(* PLC project Unnamed, Unknown Unnamed 1 *)
(* stored: creationDateTime 2025-10-15T14:42:18, modificationDateTime 2025-10-31T16:00:33 *)

(* Infeed & Conveying *)
PROGRAM program1
  VAR
    EStop AT %IX1.0 : BOOL;
    Bottle_Jam AT %IX1.1 : BOOL;  (* Sensor that monitors bottle jam. *)
    Speed_Encoder AT %IX1.2 : BOOL;  (* Conveyor speed encoder. *)
    Speed_Control AT %IX1.3 : BOOL;  (* Speed control input. *)
    Conveyor_Enable AT %MX1.0 : BOOL;  (* Memory for enabling conveyor output. *)
    Conveyor_Motor AT %QX1.0 : BOOL;  (* Conveyor motor output. *)
    Alarm_Jam AT %QX1.1 : BOOL;  (* Alarm that sounds when jam occurs. *)
    Conveyor_Speed_Command AT %QX1.2 : BOOL;  (* Output command that controls conveyor speed. *)
    Line_Light_Tower AT %QX1.3 : BOOL;  (* Indicator light for conveyor status. *)
  END_VAR

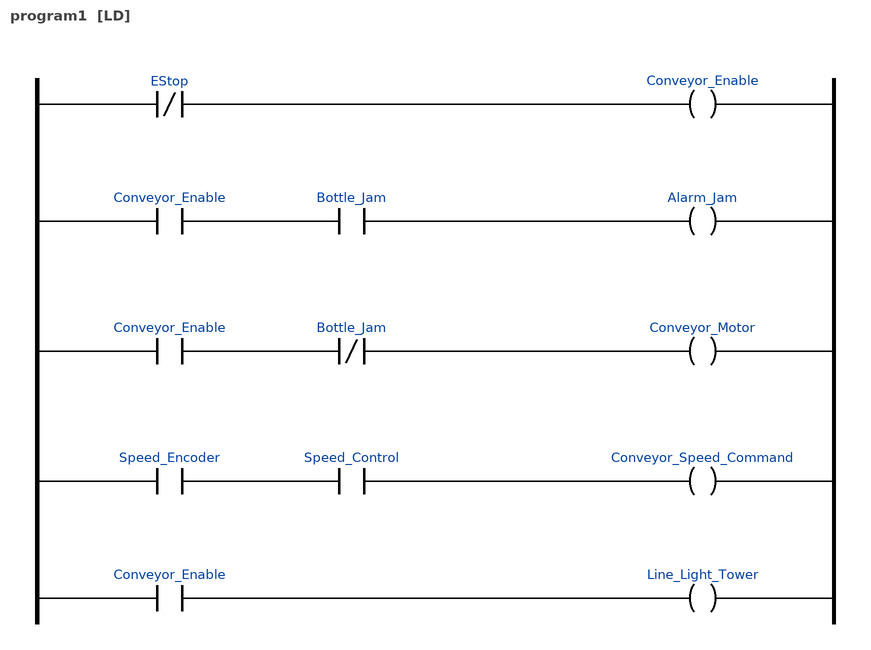
(* LD diagram, written out as Structured Text *)
Conveyor_Enable := NOT EStop;
Alarm_Jam := Conveyor_Enable AND Bottle_Jam;
Conveyor_Motor := Conveyor_Enable AND NOT Bottle_Jam;
Conveyor_Speed_Command := Speed_Encoder AND Speed_Control;
Line_Light_Tower := Conveyor_Enable;
END_PROGRAM

(* Bottle Positioning & Detection *)
PROGRAM program2
  VAR
    Switch_Conveyor AT %IX2.0 : BOOL;  (* Input switch that designates conveyor can start. *)
    Bottle_Presence_Fill AT %IX2.1 : BOOL;  (* Input that designates bottle is at filling station. *)
    Bottle_Presence_Cap AT %IX2.2 : BOOL;  (* Input that designates bottle is at capping station. *)
    Bottle_Presence_Label AT %IX2.3 : BOOL;  (* Input that designates bottle is at labeling station. *)
    Stop_Conveyor_Fill AT %MX2.0 : BOOL;  (* Stop the conveyor at the filling station. *)
    Stop_Conveyor_Cap AT %MX2.1 : BOOL;  (* Stop the conveyor at the capping station. *)
    Stop_Conveyor_Label AT %MX2.2 : BOOL;  (* Stop the conveyor at the labeling station. *)
    Conveyor_Enable AT %QX2.0 : BOOL;  (* Conveyor output. *)
  END_VAR

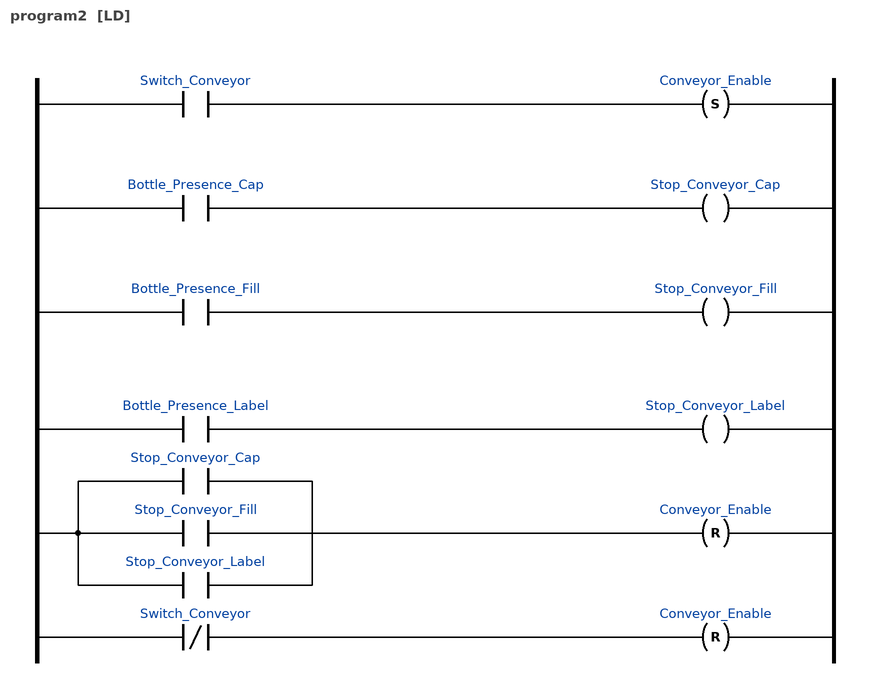
(* LD diagram, written out as Structured Text *)
Stop_Conveyor_Cap := Bottle_Presence_Cap;
Stop_Conveyor_Fill := Bottle_Presence_Fill;
Stop_Conveyor_Label := Bottle_Presence_Label;
IF Stop_Conveyor_Cap OR Stop_Conveyor_Fill OR Stop_Conveyor_Label THEN Conveyor_Enable := FALSE; END_IF;
IF Switch_Conveyor THEN Conveyor_Enable := TRUE; END_IF;
IF NOT Switch_Conveyor THEN Conveyor_Enable := FALSE; END_IF;
END_PROGRAM

(* Filling Subsystem *)
PROGRAM program3
  VAR
    Bottle_Presence_Fill AT %IX3.0 : BOOL;  (* Input that designates bottle is at filling station. *)
    Optical_Neck_Sensor AT %IX3.1 : BOOL;  (* Input that checks if bottle is okay to fill. *)
    Fill_Timer AT %IX3.2 : BOOL;  (* Input timer that tells system how long to fill bottle to full. *)
    Fill_Flowrate AT %IX3.3 : BOOL;  (* Input sensor that monitors flowrate into bottle. *)
    Fill_Temperature AT %IX3.4 : BOOL;  (* Input sensor that monitors temperature of liquid into bottle. *)
    Fill_Enable AT %MX3.0 : BOOL;  (* Memory that stores if its okay to fill. *)
    Fill_Valve AT %QX3.0 : BOOL;  (* Output fill valve. *)
    Fill_Pump_Speed AT %QX3.1 : BOOL;  (* Output fill pump speed. *)
    Fill_Alarm AT %QX3.2 : BOOL;  (* Alarm that sounds when bottle fill goes wrong. *)
  END_VAR

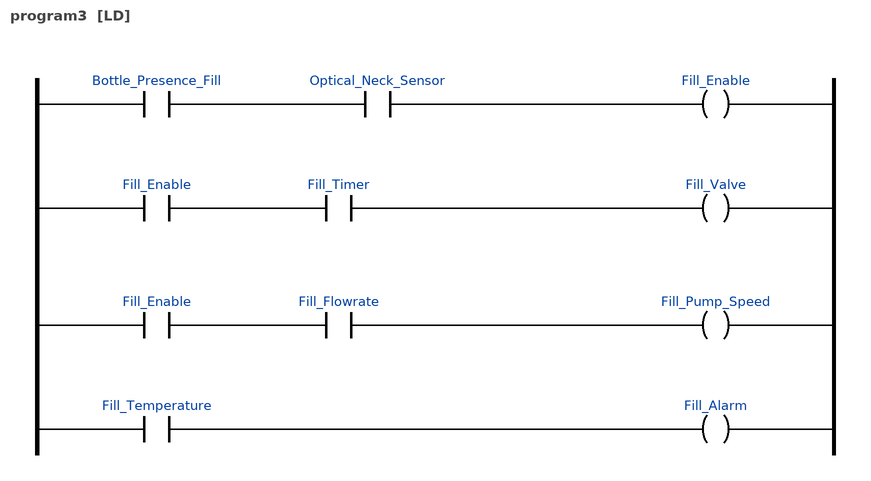
(* LD diagram, written out as Structured Text *)
Fill_Enable := Bottle_Presence_Fill AND Optical_Neck_Sensor;
Fill_Valve := Fill_Enable AND Fill_Timer;
Fill_Pump_Speed := Fill_Enable AND Fill_Flowrate;
Fill_Alarm := Fill_Temperature;
END_PROGRAM

(* Pump & Fluid Utilities *)
PROGRAM program4
  VAR
    Min_Tank_Level AT %IX4.0 : BOOL;  (* Input that arbitrates the minimum tank level. *)
    Prssure_Pump AT %IX4.1 : BOOL;  (* Input that acts as a pressure control. *)
    Pump_Enable AT %MX4.0 : BOOL;  (* Memory that stores if its okay to pump. *)
    Fill_Pump_Speed AT %QX4.0 : BOOL;  (* Output fill pump speed. *)
    Tank_Alarm AT %QX4.1 : BOOL;  (* Alarm that sounds when tank is not at optimal conditions. *)
  END_VAR

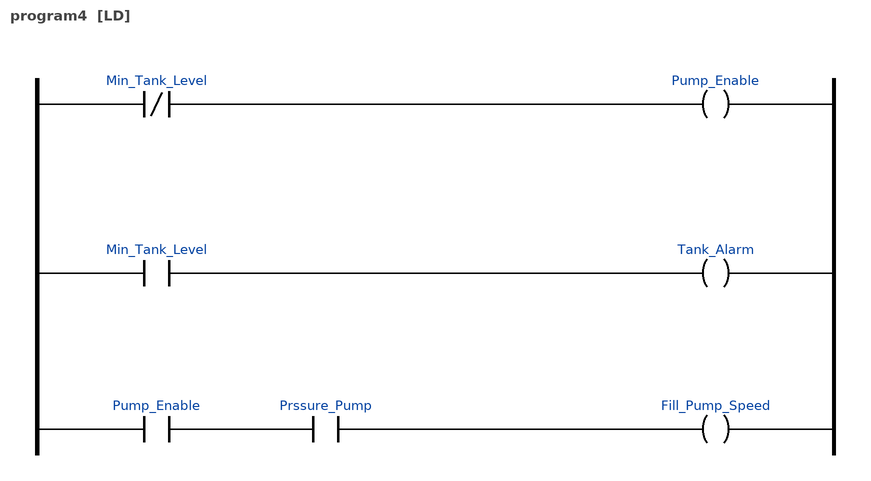
(* LD diagram, written out as Structured Text *)
Pump_Enable := NOT Min_Tank_Level;
Fill_Pump_Speed := Pump_Enable AND Prssure_Pump;
Tank_Alarm := Min_Tank_Level;
END_PROGRAM

PROGRAM program5
  VAR
    Min_Cap_Hopper_Level AT %IX5.0 : BOOL;  (* Input that determines if the cap level within the hopper is above the minium allowed amount *)
    Cap_Presence_Hopper AT %IX5.1 : BOOL;  (* Input that designates a cap is at the hopper *)
    Min_Cap_Torque_Sensor AT %IX5.2 : BOOL;  (* Input that determines if the cap torque sensor is within maximum specification *)
    Max_Cap_Torque_Sensor AT %IX5.3 : BOOL;  (* Input that determines if the cap torque sensor is within minimum specification *)
    Capping_Enable AT %MX5.0 : BOOL;  (* Memory that stores if it is okay to cap *)
    Alarm_Caps AT %QX5.1 : BOOL;  (* Alarm to notify that cap hopper level is low *)
    Cap_Bottle AT %QX5.2 : BOOL;  (* Output Capping Bottle *)
    Actuator_Alarm AT %QX5.3 : BOOL;  (* Alarm to notify if the actuator is out of specification *)
  END_VAR

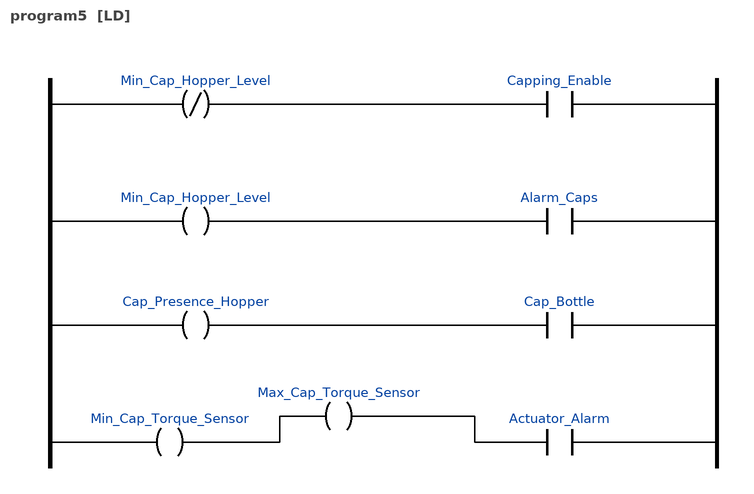
(* LD diagram, written out as Structured Text *)
Cap_Presence_Hopper := TRUE;
Min_Cap_Hopper_Level := NOT TRUE;
Min_Cap_Hopper_Level := TRUE;
Min_Cap_Torque_Sensor := TRUE;
Max_Cap_Torque_Sensor := TRUE;
(* drawn but not wired to any output: Capping_Enable, Alarm_Caps, Cap_Bottle, Actuator_Alarm *)
END_PROGRAM

PROGRAM program6
  VAR
    Bottle_Presence_Label AT %IX6.0 : BOOL;  (* Input that designates a bottle is at the labeling station *)
    Label_Presence AT %IX6.1 : BOOL;  (* Input that indicates a label is present at the labeling station *)
    Label_Positioning AT %IX6.2 : BOOL;  (* Input that checks the positioning of the label to ensure it is applied properly *)
    Label_Applicator AT %QX6.0 : BOOL;  (* Output for application of the label on to the bottle *)
    Actuator_Alarm AT %QX6.1 : BOOL;  (* Alarm to notify if the actuator is out of specification *)
  END_VAR

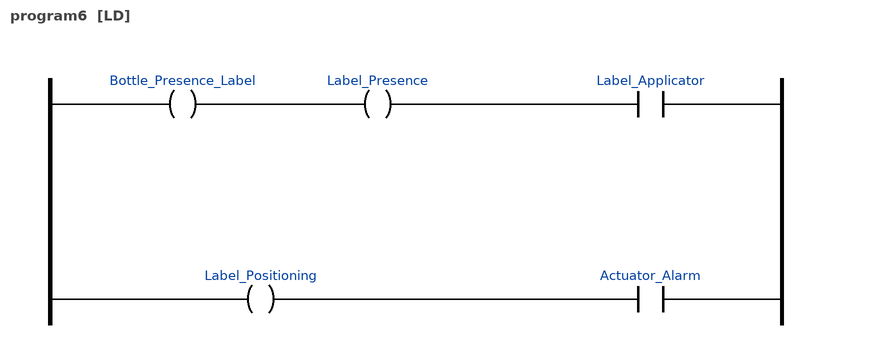
(* LD diagram, written out as Structured Text *)
Bottle_Presence_Label := TRUE;
Label_Presence := TRUE;
Label_Positioning := TRUE;
(* drawn but not wired to any output: Label_Applicator, Actuator_Alarm *)
END_PROGRAM

PROGRAM program7
  VAR
    Fill_Level_Detect AT %IX7.0 : BOOL;  (* Input to detect the level that the bottle has been filled to to ensure it is within specification *)
    Optical_Neck_sensor AT %IX7.1 : BOOL;  (* Input to detect the condition of the neck, ensuring there are no cracks or damage present on the bottle neck *)
    Bottle_Weight AT %IX7.2 : BOOL;  (* Input to detect the weight of the bottle does not exceed the threshold *)
    Cap_Torque_Sensor AT %IX7.3 : BOOL;  (* Input to detect the cap is not overtorqued *)
    Reject_Bottle AT %QX7.0 : BOOL;  (* Output to reject bottle if any of the inputs detect faults *)
  END_VAR

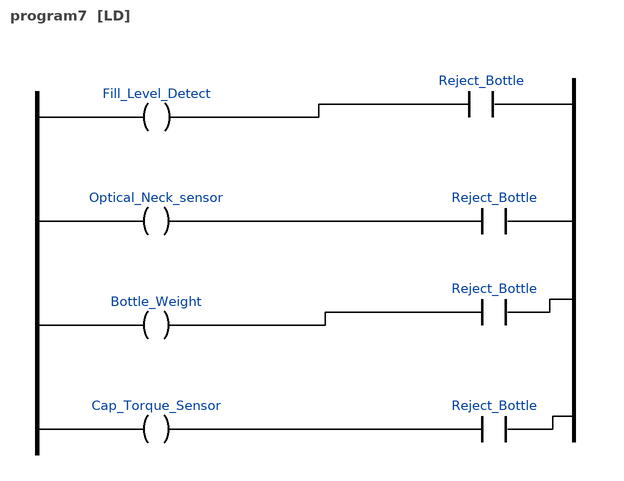
(* LD diagram, written out as Structured Text *)
Fill_Level_Detect := TRUE;
Optical_Neck_sensor := TRUE;
Bottle_Weight := TRUE;
Cap_Torque_Sensor := TRUE;
(* drawn but not wired to any output: Reject_Bottle, Reject_Bottle, Reject_Bottle, Reject_Bottle *)
END_PROGRAM

CONFIGURATION Config0
  RESOURCE Res0 ON PLC
    TASK task1(INTERVAL := T#20ms, PRIORITY := 0);
    TASK task2(INTERVAL := T#20ms, PRIORITY := 0);
    TASK task3(INTERVAL := T#20ms, PRIORITY := 0);
    TASK task4(INTERVAL := T#20ms, PRIORITY := 0);
    PROGRAM instance1 WITH task1 : program1;
    PROGRAM instance2 WITH task2 : program2;
    PROGRAM instance3 WITH task3 : program3;
    PROGRAM instance4 WITH task4 : program4;
  END_RESOURCE
END_CONFIGURATION
